// TIA Portal V20 export
TYPE "LER_typeMotionToPLC"
// stored: Access Published
   STRUCT
      Status : Struct
         Dancer : Struct
            StopRequest : Bool;
            Busy : Struct
               TotalBusy : Bool;
               EnableBusy : Bool;
               StopBusy : Bool;
               ResetBusy : Bool;
            END_STRUCT;
            Done : Struct
               TotalDone : Bool;
               EnableDone : Bool;
               StopDone : Bool;
               ResetDone : Bool;
            END_STRUCT;
            Error : Bool;
            ErrorID : DWord;
            NowCmd : DInt;
            BeforeCmd : DInt;
            NowStep : DInt;
            BeforeStep : DInt;
         END_STRUCT;
         StackMain : Struct
            StopRequest : Bool;
            Busy : Struct
               TotalBusy : Bool;
               CalculateBusy : Bool;
               SemiStepBusy : Bool;
               FullStepBusy : Bool;
               AutoBusy : Bool;
               CycleStopBusy : Bool;
               FastStopBusy : Bool;
               ResetBusy : Bool;
            END_STRUCT;
            Done : Struct
               TotalDone : Bool;
               CalculateDone : Bool;
               SemiStepDone : Bool;
               FullStepDone : Bool;
               AutoDone : Bool;
               CycleStopDone : Bool;
               FastStopDone : Bool;
               ResetDone : Bool;
            END_STRUCT;
            Error : Bool;
            ErrorID : DWord;
            NowCmd : DInt;
            BeforeCmd : DInt;
            NowStep : DInt;
            BeforeStep : DInt;
         END_STRUCT;
         OutputBits : Struct
            AnodePnP1Suction : Bool := FALSE;
            AnodePnP1Blow : Bool := FALSE;
            AnodePnP1ReelCutBlow : Bool := FALSE;
            AnodePnP1RotaryWork : Bool := FALSE;
            AnodePnP1RotaryHome : Bool := FALSE;
            AnodeReelCutDataDelete : Bool := FALSE;
            AnodePnP2Suction : Bool := FALSE;
            AnodePnP2Blow : Bool := FALSE;
            AnodeAlignSuction : Bool := FALSE;
            AnodeAlignBlow : Bool := FALSE;
            AnodeAlignVision : Bool := FALSE;
            CathodePnP1Suction : Bool := FALSE;
            CathodePnP1Blow : Bool := FALSE;
            CathodePnP1ReelCutBlow : Bool := FALSE;
            CathodePnP1RotaryWork : Bool := FALSE;
            CathodePnP1RotaryHome : Bool := FALSE;
            CathodeReelCutDataDelete : Bool := FALSE;
            CathodePnP2Suction : Bool := FALSE;
            CathodePnP2Blow : Bool := FALSE;
            CathodeAlignSuction : Bool := FALSE;
            CathodeAlignBlow : Bool := FALSE;
            CathodeAlignVision : Bool := FALSE;
            StackTableZAnodeDown : Bool := FALSE;
            StackTableZCathodeDown : Bool := FALSE;
            StackAnodeVision : Bool := FALSE;
            StackCathodeVision : Bool := FALSE;
         END_STRUCT;
         OutputData : Struct
            StackCellCount : DInt;
         END_STRUCT;
         Interface : Struct
            AutoStandby : Bool;
            AnodeReelcutStart : Bool;
            CathodeReelcutStart : Bool;
         END_STRUCT;
      END_STRUCT;
   END_STRUCT;
END_TYPE
